FUNCTION_BLOCK ILOCK_CONFLICT_TRIP_PROTECT (* Prioritizes the first active input and trips on conflict (requires RESET), with a configurable dead-time (DT_PROTECT) after release before a new direction can be activated. *)
  (* Standard: 61499-2; Description: Copyright (c) 2026 Meisterschulen am Ostbahnhof This program and the accompanying materials are made available under the terms of the Eclipse Public License 2.0 which is available at https://www.eclipse.org/legal/epl-2.0/ SPDX-License-Identifier: EPL-2.0 *)
  (* Version 1.0, 2026-09-07, Franz Höpfinger, Meisterschulen am Ostbahnhof, ILOCK_CONFLICT_TRIP + Totzeit nach Freigabe, wie ILOCK_BLOCK_PROTECT sie fuer ILOCK_BLOCK ergaenzt - TRAINING_GAPS.md Punkt 6 *)
  PACKAGE logiBUS::signalprocessing::interlock;
  (* Documentation:
  ILOCK_CONFLICT_TRIP + Dead-Time
   Kombiniert ILOCK_CONFLICT_TRIP (First-Wins, TRIP bei Konflikt, RESET nötig) mit der Schutz-Totzeit (DT_PROTECT) von ILOCK_BLOCK_PROTECT: nach Freigabe des aktiven Eingangs wird DT_PROTECT abgewartet, bevor eine neue Richtung (oder erneut ein TRIP, falls währenddessen der andere Eingang aktiviert wurde) übernommen wird.
   Unterschied zu ILOCK_CONFLICT_TRIP
   ILOCK_CONFLICT_TRIP reagiert sofort auf Freigabe des aktiven Eingangs (kein Schutzzeit-Zustand). Dieser Baustein fügt - analog zu ILOCK_BLOCK_PROTECT gegenüber ILOCK_BLOCK - die Zustände UP_STOP/DOWN_STOP ein: nach Freigabe läuft timeOut (DT_PROTECT), erst danach (Zustand EVAL) wird der tatsächlich aktuelle Zustand von DI_UP/DI_DOWN neu bewertet - inklusive TRIP, falls beide während der Totzeit aktiv wurden.
   Die TRIP-Semantik selbst (Konflikt löst sofort TRIP aus, unabhängig von der Totzeit; RESET nur akzeptiert, wenn beide Eingänge inaktiv sind) bleibt unverändert gegenüber ILOCK_CONFLICT_TRIP.
  *)
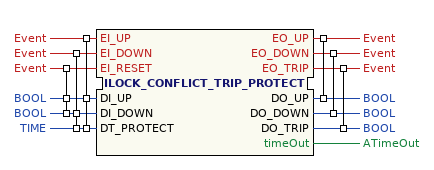
  EVENT_INPUT
    EI_UP WITH DI_UP, DT_PROTECT;
    EI_DOWN WITH DI_DOWN, DT_PROTECT;
    EI_RESET WITH DI_UP, DI_DOWN;
  END_EVENT
  EVENT_OUTPUT
    EO_UP WITH DO_UP;
    EO_DOWN WITH DO_DOWN;
    EO_TRIP WITH DO_TRIP;
  END_EVENT
  VAR_INPUT
    DI_UP : BOOL; (* TRUE = forward, up, right, clockwise *)
    DI_DOWN : BOOL; (* TRUE = backward, down, left, counter-clockwise *)
    DT_PROTECT : TIME := T#50ms; (* Protection Time *)
  END_VAR
  VAR_OUTPUT
    DO_UP : BOOL; (* TRUE = forward, up, right, clockwise *)
    DO_DOWN : BOOL; (* TRUE = backward, down, left, counter-clockwise *)
    DO_TRIP : BOOL; (* TRUE = Conflict/Trip state active *)
  END_VAR
  PLUGS
    timeOut : iec61499::events::ATimeOut; (* timeOut Adapter *)
  END_PLUGS
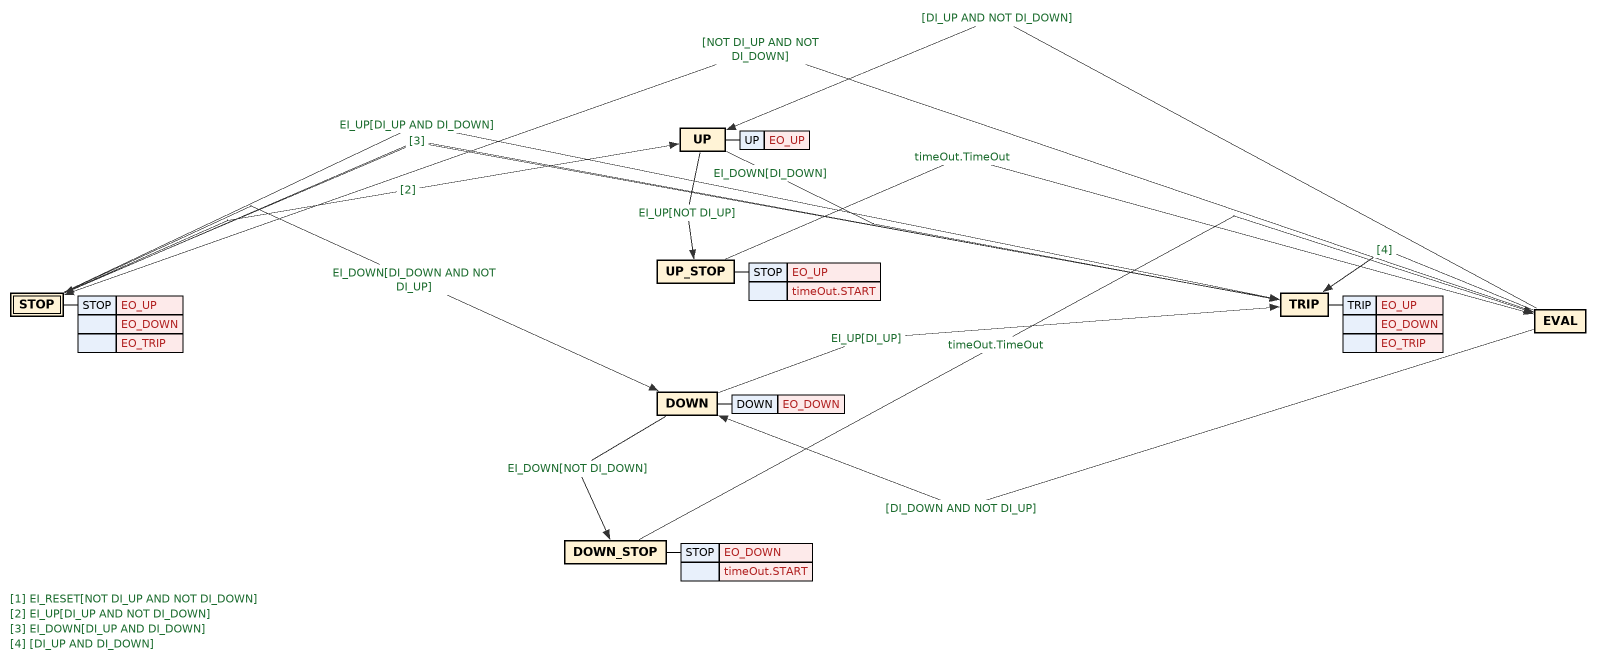
  EC_STATES
    STOP : STOP -> EO_UP, -> EO_DOWN, -> EO_TRIP;
    UP : UP -> EO_UP;
    DOWN : DOWN -> EO_DOWN;
    TRIP : TRIP -> EO_UP, -> EO_DOWN, -> EO_TRIP;
    UP_STOP : STOP -> EO_UP, -> timeOut.START;
    DOWN_STOP : STOP -> EO_DOWN, -> timeOut.START;
    EVAL;
  END_STATES
  EC_TRANSITIONS
    STOP TO UP := EI_UP[DI_UP AND NOT DI_DOWN];
    STOP TO DOWN := EI_DOWN[DI_DOWN AND NOT DI_UP];
    STOP TO TRIP := EI_UP[DI_UP AND DI_DOWN];
    STOP TO TRIP := EI_DOWN[DI_UP AND DI_DOWN];
    UP TO UP_STOP := EI_UP[NOT DI_UP];
    UP TO TRIP := EI_DOWN[DI_DOWN];
    DOWN TO DOWN_STOP := EI_DOWN[NOT DI_DOWN];
    DOWN TO TRIP := EI_UP[DI_UP];
    UP_STOP TO EVAL := timeOut.TimeOut;
    DOWN_STOP TO EVAL := timeOut.TimeOut;
    EVAL TO UP := [DI_UP AND NOT DI_DOWN];
    EVAL TO DOWN := [DI_DOWN AND NOT DI_UP];
    EVAL TO STOP := [NOT DI_UP AND NOT DI_DOWN];
    EVAL TO TRIP := [DI_UP AND DI_DOWN];
    TRIP TO STOP := EI_RESET[NOT DI_UP AND NOT DI_DOWN];
  END_TRANSITIONS
  ALGORITHM UP IN ST:
timeOut.DT := DT_PROTECT;
DO_UP := BOOL#TRUE;
DO_DOWN := BOOL#FALSE;
DO_TRIP := BOOL#FALSE;
  END_ALGORITHM
  ALGORITHM DOWN IN ST:
timeOut.DT := DT_PROTECT;
DO_UP := BOOL#FALSE;
DO_DOWN := BOOL#TRUE;
DO_TRIP := BOOL#FALSE;
  END_ALGORITHM
  ALGORITHM STOP IN ST:
timeOut.DT := DT_PROTECT;
DO_UP := BOOL#FALSE;
DO_DOWN := BOOL#FALSE;
DO_TRIP := BOOL#FALSE;
  END_ALGORITHM
  ALGORITHM TRIP IN ST:
DO_UP := BOOL#FALSE;
DO_DOWN := BOOL#FALSE;
DO_TRIP := BOOL#TRUE;
  END_ALGORITHM
END_FUNCTION_BLOCK
